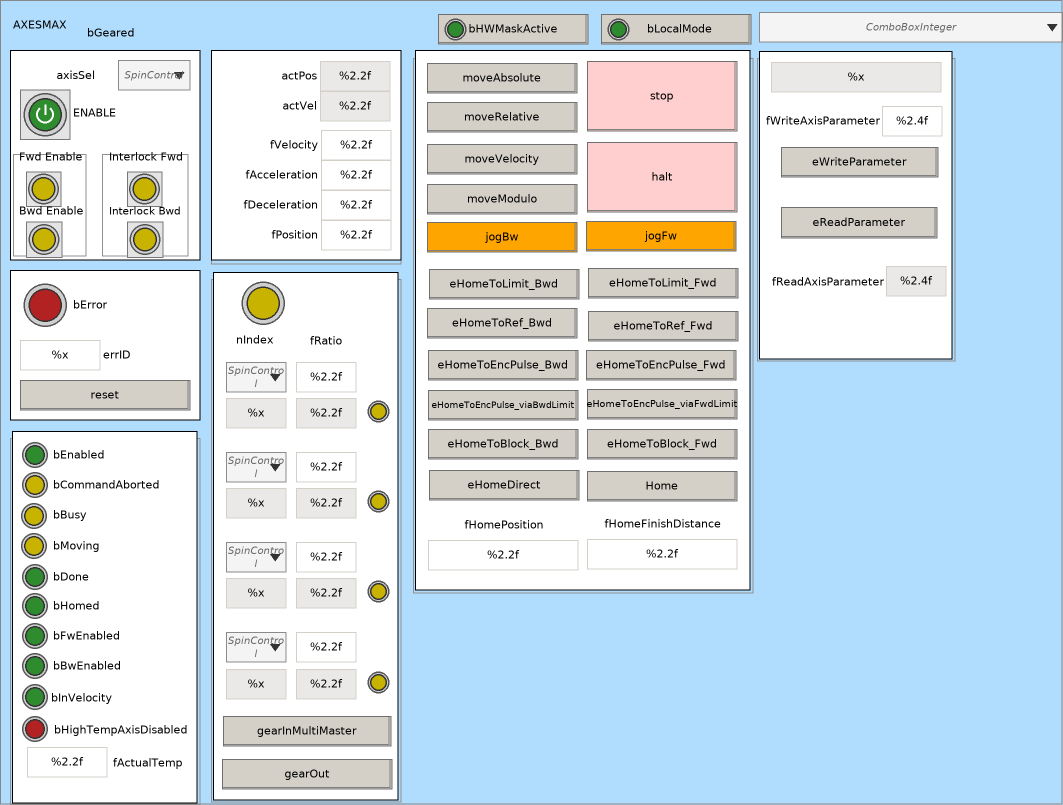
VISUALIZATION MainVisu  // 1063x805
    GroupBox (757,50 198x311)
        Rectangle (2,1 193x308)
        Textfield (14,12 170x30), "%x", text variable: astAxes[MAIN.hmiAxisSelection].stConfig.eAxisParameters
            OnMouseClick: write GVL.astAxes[MAIN.hmiAxisSelection].stConfig.eAxisParameters via Default
        Textfield (6,56 120x30), "fWriteAxisParameter", text list: "languageSupport", text index: "fWriteAxisParameter"
        Textfield (125,56 60x30), "%2.4f", text variable: astAxes[MAIN.hmiAxisSelection].stConfig.fWriteAxisParameter
            OnMouseClick: write GVL.astAxes[MAIN.hmiAxisSelection].stConfig.fWriteAxisParameter via Default
        Button (24,97 157x30), "eWriteParameter", input disabled if: GVL.astAxes[MAIN.hmiAxisSelection].stStatus.bGeared, text list: "languageSupport", text index: "eWriteParameter"
            OnMouseClick: execute { GVL.astAxes[MAIN.hmiAxisSelection].stControl.eCommand:=E_MotionFunctions.eWriteParameter; GVL.astAxes[MAIN.hmiAxisSelection].stControl.bExecute:=TRUE; }
        Button (24,157 156x31), "eReadParameter", input disabled if: GVL.astAxes[MAIN.hmiAxisSelection].stStatus.bGeared, text list: 'languageSupport', text index: "eReadParameter"
            OnMouseClick: execute { GVL.astAxes[MAIN.hmiAxisSelection].stControl.eCommand:=E_MotionFunctions.eReadParameter; GVL.astAxes[MAIN.hmiAxisSelection].stControl.bExecute:=TRUE; }
        Textfield (10,217 120x30), "fReadAxisParameter", text list: "languageSupport", text index: "fReadAxisParameter"
        Textfield (129,216 60x30), "%2.4f", text variable: astAxes[MAIN.hmiAxisSelection].stConfig.fReadAxisParameter
            OnMouseClick: write GVL.astAxes[MAIN.hmiAxisSelection].stConfig.fReadAxisParameter via Default
    GroupBox (413,50 340x543)
        Rectangle (2,0 335x540)
        Button (174,92 150x70), "halt", pressed state: GVL.astAxes[Main.hmiAxisSelection].stControl.bHalt, input disabled if: GVL.astAxes[MAIN.hmiAxisSelection].stStatus.bGeared, text list: "languageSupport", text index: "halt"
            toggle GVL.astAxes[Main.hmiAxisSelection].stControl.bHalt
        Button (174,421 150x30), "Home", input disabled if: GVL.astAxes[MAIN.hmiAxisSelection].stStatus.bGeared, text list: 'languageSupport', text index: "Home"
            OnMouseClick: execute { GVL.astAxes[Main.hmiAxisSelection].stControl.eCommand:=E_MotionFunctions.eHome; GVL.astAxes[Main.hmiAxisSelection].stControl.bExecute:=TRUE; }
        Button (15,379 150x30), "eHomeToBlock_Bwd", input disabled if: GVL.astAxes[MAIN.hmiAxisSelection].stStatus.bGeared, text list: 'languageSupport', text index: "eHomeToBlock_Bwd"
            OnMouseClick: execute {
                GVL.astAxes[Main.hmiAxisSelection].stControl.eCommand:=E_MotionFunctions.eHome;
                GVL.astAxes[Main.hmiAxisSelection].stConfig.eHomeSeq:=E_HomingRoutines.eHomeToBlock_Bwd;
                GVL.astAxes[Main.hmiAxisSelection].stControl.bExecute:=TRUE;
            }
        Button (14,258 150x30), "eHomeToRef_Bwd", input disabled if: GVL.astAxes[MAIN.hmiAxisSelection].stStatus.bGeared, text list: 'languageSupport', text index: "eHomeToRef_Bwd"
            OnMouseClick: execute {
                GVL.astAxes[Main.hmiAxisSelection].stControl.eCommand:=E_MotionFunctions.eHome;
                GVL.astAxes[Main.hmiAxisSelection].stConfig.eHomeSeq:=E_HomingRoutines.eHomeToRef_Bwd;
                GVL.astAxes[Main.hmiAxisSelection].stControl.bExecute:=TRUE;
            }
        Button (14,13 150x30), "moveAbsolute", text list: "languageSupport", text index: "moveAbsolute"
            OnMouseClick: execute { GVL.astAxes[MAIN.hmiAxisSelection].stControl.eCommand:=E_MotionFunctions.eMoveAbsolute; GVL.astAxes[MAIN.hmiAxisSelection].stControl.bExecute:=TRUE; }
        Button (14,94 150x30), "moveVelocity", input disabled if: GVL.astAxes[MAIN.hmiAxisSelection].stStatus.bGeared, text list: "languageSupport", text index: "moveVelocity"
            OnMouseClick: execute { GVL.astAxes[Main.hmiAxisSelection].stControl.eCommand:=E_MotionFunctions.eMoveVelocity; GVL.astAxes[Main.hmiAxisSelection].stControl.bExecute:=TRUE; }
        Button (14,52 150x30), "moveRelative", input disabled if: GVL.astAxes[MAIN.hmiAxisSelection].stStatus.bGeared, text list: "languageSupport", text index: "moveRelative"
            OnMouseClick: execute { GVL.astAxes[Main.hmiAxisSelection].stControl.eCommand:=E_MotionFunctions.eMoveRelative; GVL.astAxes[Main.hmiAxisSelection].stControl.bExecute:=TRUE; }
        Button (14,134 150x30), "moveModulo", input disabled if: GVL.astAxes[MAIN.hmiAxisSelection].stStatus.bGeared, text list: "languageSupport", text index: "moveModulo"
            OnMouseClick: execute { GVL.astAxes[Main.hmiAxisSelection].stControl.eCommand:=E_MotionFunctions.eMoveModulo; GVL.astAxes[Main.hmiAxisSelection].stControl.bExecute:=TRUE; }
        Button (174,11 150x70), "stop", pressed state: GVL.astAxes[Main.hmiAxisSelection].stControl.bStop, input disabled if: GVL.astAxes[MAIN.hmiAxisSelection].stStatus.bGeared, text list: "languageSupport", text index: "stop"
            toggle GVL.astAxes[Main.hmiAxisSelection].stControl.bStop
        Button (14,172 150x30), "jogBw", text list: "languageSupport", text index: "jogBw"
            OnMouseClick: execute {  }
            OnMouseDown: execute {
                GVL.astAxes[Main.hmiAxisSelection].stControl.eCommand:=E_MotionFunctions.eMoveVelocity;
                GVL.astAxes[Main.hmiAxisSelection].stControl.fVelocity:=-ABS(GVL.astAxes[Main.hmiAxisSelection].stControl.fJogVelocity)
                GVL.astAxes[Main.hmiAxisSelection].stControl.bExecute:= TRUE;
            }
            OnMouseUp: execute { GVL.astAxes[Main.hmiAxisSelection].stControl.bHalt:= TRUE; }
        Button (173,171 150x30), "jogFw", text list: "languageSupport", text index: "jogFw"
            OnMouseClick: execute {  }
            OnMouseDown: execute {
                GVL.astAxes[Main.hmiAxisSelection].stControl.eCommand:=E_MotionFunctions.eMoveVelocity;
                GVL.astAxes[Main.hmiAxisSelection].stControl.fVelocity:=ABS(GVL.astAxes[Main.hmiAxisSelection].stControl.fJogVelocity)
                GVL.astAxes[Main.hmiAxisSelection].stControl.bExecute:= TRUE;
            }
            OnMouseUp: execute { GVL.astAxes[Main.hmiAxisSelection].stControl.bHalt:= TRUE; }
        Button (175,261 150x30), "eHomeToRef_Fwd", input disabled if: GVL.astAxes[MAIN.hmiAxisSelection].stStatus.bGeared, text list: "languageSupport", text index: "eHomeToRef_Fwd"
            OnMouseClick: execute {
                GVL.astAxes[Main.hmiAxisSelection].stControl.eCommand:=E_MotionFunctions.eHome;
                GVL.astAxes[Main.hmiAxisSelection].stConfig.eHomeSeq:=E_HomingRoutines.eHomeToRef_Fwd;
                GVL.astAxes[Main.hmiAxisSelection].stControl.bExecute:=TRUE;
            }
        Button (175,218 150x30), "eHomeToLimit_Fwd", input disabled if: GVL.astAxes[MAIN.hmiAxisSelection].stStatus.bGeared, text list: "languageSupport", text index: "eHomeToLimit_Fwd"
            OnMouseClick: execute {
                GVL.astAxes[Main.hmiAxisSelection].stControl.eCommand:=E_MotionFunctions.eHome;
                GVL.astAxes[Main.hmiAxisSelection].stConfig.eHomeSeq:=E_HomingRoutines.eHomeToLimit_Fwd;
                GVL.astAxes[Main.hmiAxisSelection].stControl.bExecute:=TRUE;
            }
        Button (16,219 150x30), "eHomeToLimit_Bwd", input disabled if: GVL.astAxes[MAIN.hmiAxisSelection].stStatus.bGeared, text list: 'languageSupport', text index: "eHomeToLimit_Bwd"
            OnMouseClick: execute {
                GVL.astAxes[Main.hmiAxisSelection].stControl.eCommand:=E_MotionFunctions.eHome;
                GVL.astAxes[Main.hmiAxisSelection].stConfig.eHomeSeq:=E_HomingRoutines.eHomeToLimit_Bwd;
                GVL.astAxes[Main.hmiAxisSelection].stControl.bExecute:=TRUE;
            }
        Button (15,300 150x30), "eHomeToEncPulse_Bwd", input disabled if: GVL.astAxes[MAIN.hmiAxisSelection].stStatus.bGeared, text list: 'languageSupport', text index: "eHomeToEncPulse_Bwd"
            OnMouseClick: execute {
                GVL.astAxes[Main.hmiAxisSelection].stControl.eCommand:=E_MotionFunctions.eHome;
                GVL.astAxes[Main.hmiAxisSelection].stConfig.eHomeSeq:=E_HomingRoutines.eHomeToEncPulse_Bwd;
                GVL.astAxes[Main.hmiAxisSelection].stControl.bExecute:=TRUE;
            }
        Button (173,300 150x30), "eHomeToEncPulse_Fwd", input disabled if: GVL.astAxes[MAIN.hmiAxisSelection].stStatus.bGeared, text list: "languageSupport", text index: "eHomeToEncPulse_Fwd"
            OnMouseClick: execute {
                GVL.astAxes[Main.hmiAxisSelection].stControl.eCommand:=E_MotionFunctions.eHome;
                GVL.astAxes[Main.hmiAxisSelection].stConfig.eHomeSeq:=E_HomingRoutines.eHomeToEncPulse_Fwd;
                GVL.astAxes[Main.hmiAxisSelection].stControl.bExecute:=TRUE;
            }
        Button (174,339 150x30), "eHomeToEncPulse_viaFwdLimit", input disabled if: GVL.astAxes[MAIN.hmiAxisSelection].stStatus.bGeared, text list: "languageSupport", text index: "eHomeToEncPulse_viaFwdLimit"
            OnMouseClick: execute {
                GVL.astAxes[Main.hmiAxisSelection].stControl.eCommand:=E_MotionFunctions.eHome;
                GVL.astAxes[Main.hmiAxisSelection].stConfig.eHomeSeq:=E_HomingRoutines.eHomeToEncPulse_viaFwdLimit;
                GVL.astAxes[Main.hmiAxisSelection].stControl.bExecute:=TRUE;
            }
        Button (15,340 150x30), "eHomeToEncPulse_viaBwdLimit", input disabled if: GVL.astAxes[MAIN.hmiAxisSelection].stStatus.bGeared, text list: 'languageSupport', text index: "eHomeToEncPulse_viaBwdLimit"
            OnMouseClick: execute {
                GVL.astAxes[Main.hmiAxisSelection].stControl.eCommand:=E_MotionFunctions.eHome;
                GVL.astAxes[Main.hmiAxisSelection].stConfig.eHomeSeq:=E_HomingRoutines.eHomeToEncPulse_viaBwdLimit;
                GVL.astAxes[Main.hmiAxisSelection].stControl.bExecute:=TRUE;
            }
        Button (174,379 150x30), "eHomeToBlock_Fwd", input disabled if: GVL.astAxes[MAIN.hmiAxisSelection].stStatus.bGeared, text list: "languageSupport", text index: "eHomeToBlock_Fwd"
            OnMouseClick: execute {
                GVL.astAxes[Main.hmiAxisSelection].stControl.eCommand:=E_MotionFunctions.eHome;
                GVL.astAxes[Main.hmiAxisSelection].stConfig.eHomeSeq:=E_HomingRoutines.eHomeToBlock_Fwd;
                GVL.astAxes[Main.hmiAxisSelection].stControl.bExecute:=TRUE;
            }
        Button (16,420 150x30), "eHomeDirect", input disabled if: GVL.astAxes[MAIN.hmiAxisSelection].stStatus.bGeared, text list: 'languageSupport', text index: "eHomeDirect"
            OnMouseClick: execute {
                GVL.astAxes[Main.hmiAxisSelection].stControl.eCommand:=E_MotionFunctions.eHome;
                GVL.astAxes[Main.hmiAxisSelection].stConfig.eHomeSeq:=E_HomingRoutines.eHomeDirect;
                GVL.astAxes[Main.hmiAxisSelection].stControl.bExecute:=TRUE;
            }
        Textfield (15,490 150x30), "%2.2f", text variable: GVL.astAxes[MAIN.hmiAxisSelection].stConfig.fHomePosition
            OnMouseClick: write the text variable via Default
        Textfield (174,489 150x30), "%2.2f", text variable: GVL.astAxes[MAIN.hmiAxisSelection].stConfig.fHomeFinishDistance, text list: ''
            OnMouseClick: write the text variable via Default
        Textfield (175,459 150x30), "fHomeFinishDistance", text list: "languageSupport", text index: "fHomeFinishDistance"
        Textfield (16,460 150x30), "fHomePosition", text list: "languageSupport", text index: "fHomePosition"
    GroupBox (211,271 190x531)
        Rectangle (2,1 185x528)
        SpinControl (15,91 60x30), variable: GVL.astAxes[MAIN.hmiAxisSelection].stConfig.astMultiMasterAxis[1].nIndex
            p651134158: GVL_APP.nAXIS_NUM
        Textfield (85,91 60x30), "%2.2f", text variable: GVL.astAxes[MAIN.hmiAxisSelection].stConfig.astMultiMasterAxis[1].fRatio
            OnMouseClick: write the text variable via Default
        Textfield (80,55 70x30), "fRatio", text list: "languageSupport", text index: "gearRatio"
        Button (12,445 168x30), "gearInMultiMaster", text list: "languageSupport", text index: "gearIn"
            OnMouseClick: execute { GVL.astAxes[Main.hmiAxisSelection].stControl.eCommand:=E_MotionFunctions.eGearInMultiMaster; GVL.astAxes[Main.hmiAxisSelection].stControl.bExecute:=TRUE; }
        SpinControl (15,181 60x30), variable: GVL.astAxes[MAIN.hmiAxisSelection].stConfig.astMultiMasterAxis[2].nIndex
            p651134158: GVL_APP.nAXIS_NUM
        SpinControl (15,271 60x30), variable: GVL.astAxes[MAIN.hmiAxisSelection].stConfig.astMultiMasterAxis[3].nIndex
            p651134158: GVL_APP.nAXIS_NUM
        SpinControl (15,361 60x30), variable: GVL.astAxes[MAIN.hmiAxisSelection].stConfig.astMultiMasterAxis[4].nIndex
            p651134158: GVL_APP.nAXIS_NUM
        Textfield (85,181 60x30), "%2.2f", text variable: GVL.astAxes[MAIN.hmiAxisSelection].stConfig.astMultiMasterAxis[2].fRatio
            OnMouseClick: write the text variable via Default
        Textfield (85,271 60x30), "%2.2f", text variable: GVL.astAxes[MAIN.hmiAxisSelection].stConfig.astMultiMasterAxis[3].fRatio
            OnMouseClick: write the text variable via Default
        Textfield (85,361 60x30), "%2.2f", text variable: GVL.astAxes[MAIN.hmiAxisSelection].stConfig.astMultiMasterAxis[4].fRatio
            OnMouseClick: write the text variable via Default
        Button (11,488 170x30), "gearOut", text list: "languageSupport", text index: "gearOut"
            OnMouseClick: execute { GVL.astAxes[Main.hmiAxisSelection].stControl.eCommand:=E_MotionFunctions.eGearOut; GVL.astAxes[Main.hmiAxisSelection].stControl.bExecute:=TRUE; }
        Textfield (9,54 70x30), "nIndex", text list: "languageSupport", text index: "masterGear"
        Textfield (85,127 60x30), "%2.2f", text variable: GVL.astAxes[MAIN.hmiAxisSelection].Axis.PlcToNc.GearRatio1
        Textfield (15,127 60x30), "%x", text variable: GVL.astAxes[MAIN.hmiAxisSelection].stConfig.astMultiMasterAxisLatched[1].nIndex
        Textfield (85,217 60x30), "%2.2f", text variable: GVL.astAxes[MAIN.hmiAxisSelection].Axis.PlcToNc.GearRatio2
        Textfield (15,217 60x30), "%x", text variable: GVL.astAxes[MAIN.hmiAxisSelection].stConfig.astMultiMasterAxisLatched[2].nIndex
        Textfield (85,307 60x30), "%2.2f", text variable: GVL.astAxes[MAIN.hmiAxisSelection].Axis.PlcToNc.GearRatio3
        Textfield (15,307 60x30), "%x", text variable: GVL.astAxes[MAIN.hmiAxisSelection].stConfig.astMultiMasterAxisLatched[3].nIndex
        Textfield (85,398 60x30), "%2.2f", text variable: GVL.astAxes[MAIN.hmiAxisSelection].Axis.PlcToNc.GearRatio4
        Textfield (15,398 60x30), "%x", text variable: GVL.astAxes[MAIN.hmiAxisSelection].stConfig.astMultiMasterAxisLatched[4].nIndex
        Lamp1 (155,399 25x25), variable: GVL.astAxes[MAIN.hmiAxisSelection].stStatus.bCoupledGear4, style: Lamp-Lamp1-Yellow
        Lamp1 (155,308 25x25), variable: GVL.astAxes[MAIN.hmiAxisSelection].stStatus.bCoupledGear3, style: Lamp-Lamp1-Yellow
        Lamp1 (155,218 25x25), variable: GVL.astAxes[MAIN.hmiAxisSelection].stStatus.bCoupledGear2, style: Lamp-Lamp1-Yellow
        Lamp1 (155,128 25x25), variable: GVL.astAxes[MAIN.hmiAxisSelection].stStatus.bCoupledGear1, style: Lamp-Lamp1-Yellow
        Lamp1 (27,7 50x50), variable: GVL.astAxes[MAIN.hmiAxisSelection].stStatus.bGeared, style: Lamp-Lamp1-Yellow
    GroupBox (10,50 190x210)
        Rectangle (0,0 190x210)
        GroupBox (3,96 73x110)
        GroupBox (92,96 86x110)
        Textfield (60,50 92x26), "ENABLE", text list: 'languageSupport', text index: "enable"
        PushSwitchLed (16,118 35x42), variable: GVL.astAxes[MAIN.hmiAxisSelection].stInputs.bLimitFwd, behaviour: TOGGLE, style: Switch-PushSwitchLed-Yellow
        PushSwitchLed (16,170 36x39), variable: GVL.astAxes[MAIN.hmiAxisSelection].stInputs.bLimitBwd, behaviour: TOGGLE, style: Switch-PushSwitchLed-Yellow
        SpinControl (108,10 72x30), variable: MAIN.hmiAxisSelection
            p651134158: GVL_APP.nAXIS_NUM
        Textfield (23,13 86x25), "axisSel", text variable: GVL_APP.nAXIS_NUM, text list: "languageSupport", text index: "axisSel"
        PowerSwitch (10,38 50x53), variable: GVL.astAxes[MAIN.hmiAxisSelection].stControl.bEnable, behaviour: TOGGLE, style: Switch-PowerSwitch-Green
        PushSwitchLed (117,118 35x42), variable: GVL.astAxes[MAIN.hmiAxisSelection].stControl.bInterlockFwd, behaviour: TOGGLE, style: Switch-PushSwitchLed-Yellow
        PushSwitchLed (117,170 36x39), variable: GVL.astAxes[MAIN.hmiAxisSelection].stControl.bInterlockBwd, behaviour: TOGGLE, style: Switch-PushSwitchLed-Yellow
        Textfield (6,94 76x26), "Fwd Enable", text list: 'languageSupport', text index: "enFW"
        Textfield (6,148 76x26), "Bwd Enable", text list: 'languageSupport', text index: "enBW"
        Textfield (96,94 76x26), "Interlock Fwd", text list: 'languageSupport', text index: "bAxisInterlockFwd"
        Textfield (96,148 76x26), "Interlock Bwd", text list: 'languageSupport', text index: "bAxisInterlockBwd"
    Textfield (10,10 231x30), "AXESMAX", text variable: GVL_APP.nAXIS_NUM, text list: "languageSupport", text index: "axesAvailable"
    GroupBox (10,270 190x150)
        Rectangle (0,0 190x150)
        Textfield (90,70 90x30), "errID", text list: "languageSupport", text index: "errID"
        Textfield (10,70 80x30), "%x", text variable: GVL.astAxes[MAIN.hmiAxisSelection].stStatus.nErrorID
        Lamp1 (10,10 50x50), variable: GVL.astAxes[MAIN.hmiAxisSelection].stStatus.bError, style: Lamp-Lamp1-Red
        Textfield (60,20 120x30), "bError", text list: "languageSupport", text index: "bError"
        Button (10,110 170x30), "reset", pressed state: GVL.astAxes[Main.hmiAxisSelection].stControl.bReset, text list: "languageSupport", text index: "reset"
            OnMouseClick: toggle GVL.astAxes[Main.hmiAxisSelection].stControl.bReset
    GroupBox (10,430 190x375)
        Rectangle (2,1 185x372)
        Lamp1 (10,10 30x30), variable: GVL.astAxes[MAIN.hmiAxisSelection].stStatus.bEnabled, style: Lamp-Lamp1-Green
        Textfield (40,10 140x30), "bEnabled", text list: "languageSupport", text index: "bEnabled"
        Lamp1 (10,40 30x30), variable: GVL.astAxes[MAIN.hmiAxisSelection].stStatus.bCommandAborted, style: Lamp-Lamp1-Yellow
        Textfield (40,40 140x30), "bCommandAborted", text list: "languageSupport", text index: "bCommandAborted"
        Textfield (40,70 140x30), "bBusy", text list: "languageSupport", text index: "bBusy"
        Lamp1 (10,132 30x30), variable: GVL.astAxes[MAIN.hmiAxisSelection].stStatus.bDone, style: Lamp-Lamp1-Green
        Textfield (40,132 140x30), "bDone", text list: 'languageSupport', text index: "bDone"
        Lamp1 (10,161 30x30), variable: GVL.astAxes[MAIN.hmiAxisSelection].stStatus.bHomed, style: Lamp-Lamp1-Green
        Textfield (40,161 140x30), "bHomed", text list: "languageSupport", text index: "bHomed"
        Lamp1 (10,191 30x30), variable: GVL.astAxes[MAIN.hmiAxisSelection].stStatus.bFwEnabled AND NOT GVL.astAxes[MAIN.hmiAxisSelection].stStatus.bInterlockedFwd, style: Lamp-Lamp1-Green
        Lamp1 (10,221 30x30), variable: GVL.astAxes[MAIN.hmiAxisSelection].stStatus.bBwEnabled AND NOT GVL.astAxes[MAIN.hmiAxisSelection].stStatus.bInterlockedBwd, style: Lamp-Lamp1-Green
        Textfield (40,191 140x30), "bFwEnabled", text list: "languageSupport", text index: "bFwEnabled"
        Textfield (40,221 140x30), "bBwEnabled", text list: "languageSupport", text index: "bBwEnabled"
        Lamp1 (9,71 30x30), variable: GVL.astAxes[MAIN.hmiAxisSelection].stStatus.bBusy, style: Lamp-Lamp1-Yellow
        Lamp1 (10,252 30x30), variable: GVL.astAxes[MAIN.hmiAxisSelection].stStatus.bInVelocity, style: Lamp-Lamp1-Green
        Lamp1 (10,284 30x30), variable: GVL.astAxes[MAIN.hmiAxisSelection].stStatus.bHighTempAxisDisabled, style: Lamp-Lamp1-Red
        Textfield (17,317 80x30), "%2.2f", text variable: GVL.astAxes[MAIN.hmiAxisSelection].stStatus.fActTemperature
        Textfield (100,318 79x30), "fActualTemp", text list: "languageSupport", text index: "fActualTemp"
        Textfield (38,253 140x30), "bInVelocity", text list: 'languageSupport', text index: "bInVelocity"
        Textfield (41,285 140x30), "bHighTempAxisDisabled", text list: 'languageSupport', text index: "bHighTempDisable"
        Lamp1 (9,101 30x30), variable: GVL.astAxes[MAIN.hmiAxisSelection].stStatus.bMoving, style: Lamp-Lamp1-Yellow
        Textfield (40,101 140x30), "bMoving", text list: "languageSupport", text index: "bMoving"
    GroupBox (211,50 190x214)
        Rectangle (0,0 190x210)
        Textfield (10,80 100x30), "fVelocity", text list: "languageSupport", text index: "fVelocity"
        Textfield (110,80 70x30), "%2.2f", text variable: GVL.astAxes[MAIN.hmiAxisSelection].stControl.fVelocity
            OnMouseClick: write the text variable via Default
        Textfield (10,110 100x30), "fAcceleration", text list: "languageSupport", text index: "fAcceleration"
        Textfield (110,110 70x30), "%2.2f", text variable: GVL.astAxes[MAIN.hmiAxisSelection].stControl.fAcceleration
            OnMouseClick: write the text variable via Default
        Textfield (10,140 100x30), "fDeceleration", text list: "languageSupport", text index: "fDeceleration"
        Textfield (110,140 70x30), "%2.2f", text variable: GVL.astAxes[MAIN.hmiAxisSelection].stControl.fDeceleration
            OnMouseClick: write the text variable via Default
        Textfield (10,170 100x30), "fPosition", text list: "languageSupport", text index: "fPosition"
        Textfield (110,170 70x30), "%2.2f", text variable: GVL.astAxes[MAIN.hmiAxisSelection].stControl.fPosition
            OnMouseClick: write the text variable via Default
        Textfield (109,11 70x30), "%2.2f", text variable: GVL.astAxes[MAIN.hmiAxisSelection].stStatus.fActPosition
        Textfield (9,11 100x30), "actPos", text list: "languageSupport", text index: "actposition"
        Textfield (9,41 100x30), "actVel", text list: "languageSupport", text index: "actVelocity"
        Textfield (109,41 70x30), "%2.2f", text variable: GVL.astAxes[MAIN.hmiAxisSelection].stStatus.fActVelocity
        Textfield (-127,-32 93x30), "bGeared", text list: "languageSupport", text index: "bGeared"
    Group (601,14 150x30)
        Button (0,0 150x30), "bLocalMode", text list: 'languageSupport', text index: 'bLocalMode'
            OnMouseClick: toggle bLocalMode
        Lamp1 (5,3 25x25), variable: bLocalMode, style: Lamp-Lamp1-Green
    ComboBoxInteger (759,12 304x30), variable: GVL.astAxes[MAIN.hmiAxisSelection].stConfig.eAxisParameters, text list: 'ParameterTextList'
    Group (438,14 150x30)
        Button (0,0 150x30), "bHWMaskActive", text list: 'languageSupport', text index: 'bHWMaskActive'
            OnMouseClick: toggle bLocalMode
        Lamp1 (5,3 25x25), variable: GVL.astAxes[MAIN.hmiAxisSelection].stControl.bHWMaskActive, style: Lamp-Lamp1-Green
END_VISUALIZATION

(* stored: Version 1.1.0.1, ProductVersion 3.1.4024.12
   Visu MainVisu: Id {98c8ae72-e756-4d11-b6a5-5914882e2424} *)
